INTERFACE ITF_GroupElement_HMI

METHOD LinkGroupelementData : BOOL
VAR_INPUT
	stData					: ST_GroupElement_HMI;
END_VAR
END_METHOD

END_INTERFACE

(* stored: Version 1.1.0.1, ProductVersion 3.1.4024.15
   Itf ITF_GroupElement_HMI: Id {56ded6a8-c57d-4918-9207-29ee5c9f0bfe}
   Method LinkGroupelementData: Id {64ef952f-6751-437c-b0de-46c34b5f4196} *)
